FUNCTION_BLOCK "fbUO_MX_SETUP"
TITLE = UO : MX_SETUP
{ S7_Optimized_Access := 'TRUE' }
AUTHOR : REO
NAME : MX_SETUP
VERSION : 2.0
//****************************************************************************************************
// Code generated by SFC Generator V1.13 on 23/11/18 15:00:24 by  David Paspa from File G:\Business\Synertec\MPI.SMS\automation\code\awlMaster\stencil\seq_hdr.awl
//****************************************************************************************************
//****************************************************************************************************
//================================ SEQ HEADER ================================//
//            Copyright 2018 Rieckermann Engineering Operations               //
//----------------------------------------------------------------------------//
// Title: UO_MX_SETUP                                                       //
//                                                                            //
// Description:                                                               //
// Unit Operation for setup of equipment for manufacturing operations.                                                        //
//                                                                            //
// // SFC Revision History:
// Rev By               Date        CC         Note
// 2.0 David Paspa      09-Aug-2018            Reboot for S7-1500.
// 0.1 Gerald Kontriner 14-Sep-2009            SFC structural design                                                       //
//----------------------------------------------------------------------------//
// Sequencer Revision History:                                                //
// Rev By               Date        CC        Note                            //
// 2.0 David Paspa      05-Jan-2018 NA        Reboot for S7-1500.             //
// 1.6 Khairul Basar    19-Nov-2009 NA        Reset #sqSequencer.STEP.Active  //
//                                            when STEP Finished.             //
// 1.5 Khairul Basar    15-Oct-2009 NA        Placeholder inserted:           //
//                                            "udtSQ_UO";          //
// 1.4 Khairul Basar    06-Oct-2009 NA        R #PAUSE;                       //
// 1.3 Khairul Basar    30-Sep-2009 NA        SEQ_HDR change STEP-0 code      //
//                                            deleted.                        //
// 1.2 Khairul Basar    26-Sep-2009 NA        Refer R4.                       //
// 1.1 Khairul Basar    23-Sep-2009 NA        Refer R3.                       //
// 1.0 Khairul Basar    20-Sep-2009 NA        STEP.Finished flag reset by     //
//                                            JUMP_MAN.                       //
// 0.9 Khairul Basar    11-Sep-2009 NA        SQ_TIMER added as VAR, declared //
//                                            in SEQ_FTR.                     //
// 0.8 Khairul Basar    09-Sep-2009 NA        SqSequencer.Err_Fault is reset  //
//                                            on Stop cmd, Step-0 dead code   //
//                                            deleted from ACT & Verify.      //
//                                            STP_FTR Step_withErr flag       //
//                                            STEP_NUM place holder           //
//                                            configured.                     //
// 0.7 Khairul Basar    28-Aug-2009 NA        SQ_FINISHED OUT added again.    //
//                                            Deleted during major mod R3.    //
// 0.6 Khairul Basar    23-Aug-2009 NA        Refer R2.                       //
// 0.5 Khairul Basar    23-Aug-2009 NA        Refer R1.                       //
// 0.4 Khairul Basar    18-Aug-2009 NA        Reset Step done with/out error  //
//                                            bits using FC:RSET.             //
// 0.3 David Paspa      16-Aug-2009 NA        Added placeholders for header   //
//                                            name and version and revision   //
//                                            history.                        //
// 0.2 Khairul Basar    11-Aug-2009 NA        Retired external udt file for   //
//                                            Static type parameters. All     //
//                                            parameters now IN, OUT or       //
//                                            IN_OUT.                         //
// 0.1 Khairul Basar    12-Jun-2009 NA        Initial design.                 //
//----------------------------------------------------------------------------//
// R4:                                                                        //
// 1.If SQ not finished Resume command will start Step timer, and redo the    //
// last action, verify the feedback.                                          //
// 2."STEP.finished" flag is ANDed with "TRN_AND_JUMP" in the snippet file    //
// TRN_HDR.This is to avoid checking of transition logic if STEP is not       //
// finished yet.                                                              //
// 3.MDCH, Load & transfer typo corrected.                                    //
//                                                                            //
// R3:                                                                        //
// 1.SqStepTimer.IN is reset in STEP_FTR instead of resetting it in TRN_HDR.  //
// This is because TRN_HDTR is not included in the Last step and StepTimer    //
// must reset in the last step.                                               //
// 2.Reset all the timers when SQ stops.Reset done in SEQ_HDR.                //
// Also STEP-finished flag reset when SQ is OFF to                            //
// scan last step.                                                            //
//                                                                            //
// R2:                                                                        //
// 1.Any step error will send the Sequencer into Pause state.Code added in    //
// SEQ_HDR.Snippet Place holder for Bool-array 24 is   //
// deleted.                                                                   //
//                                                                            //
// R1:                                                                        //
// 1.sqStepTimer:All Verification Code must satisfy the condition finish step //
// action within STEP_DELAY time(40s).If step actions not finished within the //
// time period the error flag will raise High signal.Else timer will reset.   //
// 2.sqRunTimer Added therefore can be used as retentive & non retentive.     //
// 3.sqSequencer: This is re-structured UDT which is redefined the symbol     //
// names as well as it gives more clearity.                                   //
// 4.fcMODE and fcCMD functions are added to handle the mode & command        //
// independently regardless of other logic.Two separate UDT udtMODE & udt     //
// CMD assigned to Mode & command function respectively.                      //
// 5.MAN_JUMP programed for manual mode jump operation with or without        //
// Transition code satisfied.TRN_AND_JUMP & NO_VERIFC are the parameters      //
// which will define whether verification code & transition code need to be   //
// checked to perform jump operation.                                         //
// 6.Auto to Manual switchover will be bumpless & will not affect step        //
// operation.Manual to auto switchover can be used to resume Step action at   //
// defined.                                                                   //
// Step number entered in STEPNO_JUMP.                                        //
//                                                                            //
// Parameters:                                                                //
// INPUTS                                                                     //
// ======                                                                     //
// SQ_CMD          Sequence command input inherited from object block         //
//                 0: off/idle                                                //
//                 1: start/initiate                                          //
//                 2: pause                                                   //
//                 3: resume                                                  //
//                 4: reserved (not programmed)                               //
//                 5: reserved (not programmed)                               //
//                 6: abort/go to last step                                   //
//                 7: acknowledge error/fault                                 //
// SQ_MODE         Sequencer Auto/Manual input inherited from object block    //
//                 1: manual                                                  //
//                 2: auto                                                    //
//                                                                            //
// INPUT/OUTPUTS                                                              //
// =============                                                              //
// SQ_JUMP_MAN     Allows manual jumping from one step to the next step. The  //
//                 manual jump flag is ORed with the transition process       //
//                 condition and so can be used to bypass the condition if the//
//                 sequence will not progress.                                //
//                 This input can also be used to jump to any step even       //
//                 when no transition -> step linkage exists. This is only    //
//                 possible when the SQ_MODE is in manual and SQ is in the    //
//                 idle step. The step to jump to is specified in             //
//                 SQ_man_jump_to_step (not accesseble by this FB in/out      //
//                 interface but a separate DB memory location).              //
//                                                                            //
// OUTPUTS                                                                    //
// =======                                                                    //
// SQ_STATE        The calculated state of the sequence                       //
//                 0: off/idle                                                //
//                 1: start/initiated                                         //
//                 2: paused                                                  //
//                 3: resumed                                                 //
//                 4: reserved (wrong Mode)                                   //
//                 5: reserved (Wrong commad)                                 //
//                 6: aborted/go to last step                                 //
//                 7: acknowledged error/fault                                //
// CURSTEP         Current step being proccessed.                             //
// S_ACTIVE        If current step is active                                  //
// NXT_STEP        Next step to jump to if transition condition is true       //
// ERR_FAULT       True if any error/ or fault present                        //
// PAUSED          True if step is paused                                     //
// OFF_IDLE        Sequence is not running but ready for next SQ (in step=0)  //
//----------------------------------------------------------------------------//
// Define variables:                                                          //
//----------------------------------------------------------------------------//
   VAR_IN_OUT
      _emm_vessel_mi_vessel_pv : Real;   // Vessel measured mass
      _emx_drain_state : Int;   // State for MX drain valves
      _emv_inlet_state : Int;   // Sprayball inlet state
      _emt_hex_state : Int;   // Heat exchanger temperature control state
      _vessel_mx : Int;   // Manufacturing vessel selection M1 or M2
      _emc_gas_pi_vessel_pv : Real;   // Vessel pressure
      _vacuum_hold_test : Bool;   // Vacuum hold test enquiry
      _emm_vessel_state : Int;   // Device State of emm_vessel
      _emc_water_state : Int;   // Device State of emc_water
      _emx_mmfl_state : Int;   // Device State of emx_mmfl
      _emv_vessel_state : Int;   // Device State of EVxy04
      _emg_filter_state : Int;   // Device State of emg_filter
      _emx_transfer_state : Int;   // Device State of emx_transfer
      _emc_gas_state : Int;   // Device State of emc_gas
      _emx_drain_subs : Int;   // Substate for MX drain valves
      _emx_drain_cmd : Int;   // Command for MX drain valves
      _emv_inlet_subs : Int;   // Sprayball inlet substate
      _emv_inlet_cmd : Int;   // Sprayball inlet command
      _emt_hex_cmd : Int;   // Heat exchanger temperature control command
      _emt_hex_subs : Int;   // Heat exchanger temperature control substate
      _emt_hex_drain_time : Time;   // Heat exchanger drain time
      _emc_gas_medium_gas : Int;   // Medium selection for emc_gas
      _emm_vessel_cmd : Int;   // Command to emm_vessel
      _emm_vessel_subs : Int;   // Substate selection to emm_vessel
      _emc_water_cmd : Int;   // Command to emc_water
      _emc_water_subs : Int;   // Substate selection to emc_water
      _emc_water_medium_liquid : Int;   // Medium selection for emc_water
      _emx_mmfl_cmd : Int;   // Command to emx_mmfl
      _emv_vessel_subs : Int;   // Substate selection to emv_vessel
      _emx_mmfl_subs : Int;   // Substate selection to emx_mmfl
      _emv_vessel_cmd : Int;   // Command to emv_vessel
      _emx_transfer_cmd : Int;   // Command to emx_transfer
      _emg_filter_cmd : Int;   // Command to emg_filter
      _emx_transfer_subs : Int;   // Substate selection to EXxy07
      _emg_filter_subs : Int;   // Substate selection to emg_filter
      _emc_gas_cmd : Int;   // Command to emc_gas
      _emc_gas_subs : Int;   // Substate selection to emc_gas
      dummy : Bool;   // Dummy placeholder for call without comma
   END_VAR

   VAR
      smc : "udtModeCommandSFC";   // SFC mode and command
      sqStepTimer {OriginalPartName := 'IEC_TIMER'; LibVersion := '1.0'} : TON_TIME;
      sqRunTimer : "fbRunTimer";
      sqSequencer : "udtSFCSequence32";
      SQ_TIMER {OriginalPartName := 'IEC_TIMER'; LibVersion := '1.0'} : TON_TIME;
      SQ_TIMER2 {OriginalPartName := 'IEC_TIMER'; LibVersion := '1.0'} : TON_TIME;
      SQ_TIMER3 {OriginalPartName := 'IEC_TIMER'; LibVersion := '1.0'} : TON_TIME;
      sqSeqTimerStart : Bool;
      sqSeqTimerStart2 : Bool;
      sqSeqTimerStart3 : Bool;
      sqSeqTimerElapsed : Time;
      sqSeqTimerElapsed2 : Time;
      sqSeqTimerElapsed3 : Time;
      sqSeqTimerExpired : Bool;
      sqSeqTimerExpired2 : Bool;
      sqSeqTimerExpired3 : Bool;
      sqStepTimerElapsed : Time;
      sqStepTimerExpired : Bool;
      _r_time_hex_drain : Time;   // MX SETUP Heat exchanger drain time
      _real_not_held : Real;   // UO_MX_SETUP Vacuum pressure hold test failed
      _real_vacuum_fail : Real;   // UO_MX_SETUP Vacuum failed pressure after vacuum timer expired
      _log_real_pressure_mx : Bool;   // UO_MX_SETUP Vessel pressure
      _real_pressure_mx : Real;   // UO_MX_SETUP Vessel pressure
      _log_real_not_held : Bool;   // UO_MX_SETUP Vacuum pressure hold test failed
      _vacuum_held_begin_time : Time_Of_Day;   // vacuum hold begin time
      _vacuum_held_end_time : Time_Of_Day;   // vacuum hold end time
      _time_act_vacuum_held : Time;   // UO_MX_SETUP Vacuum held time
      _log_time_act_vacuum_held : Bool;   // UO_MX_SETUP Vacuum held time
      _prompt_not_held : Bool;   // UO_MX_SETUP Operator to confirm to retry as vacuum pressure not held
      _prompt_not_held_confirm_yes : Bool;   // UO_MX_SETUP Operator to confirm to retry vacuum pressure not held confirmed yes
      _prompt_not_held_confirm_no : Bool;   // UO_MX_SETUP Operator to confirm to retry vacuum pressure not held confirmed no
      _log_msg_not_held_repeat : Bool;   // UO_MX_SETUP Operator confirmed to retry when vacuum pressure not held
      _log_msg_not_held_abort : Bool;   // UO_MX_SETUP Operator confirmed to abort when vacuum pressure not held
      _prompt_not_reach : Bool;   // UO_MX_SETUP Operator to confirm retry when vacuum pressure not reached setpoint
      _prompt_not_reach_confirm_yes : Bool;   // UO_MX_SETUP Operator confirmed retry when vacuum pressure not reached setpoint
      _prompt_not_reach_confirm_no : Bool;   // UO_MX_SETUP Operator confirmed abort when vacuum pressure not reached setpoint
      _log_msg_not_reach_repeat : Bool;   // UO_MX_SETUP Operator confirmed retry when vacuum pressure not reached setpoint
      _log_msg_not_reach_abort : Bool;   // UO_MX_SETUP Operator confirmed abort when vacuum pressure not reached setpoint
      _log_real_vacuum_fail : Bool;   // UO_MX_SETUP Vacuum failed after vacuum timer expired
      _log_msg_vacuum_begin : Bool;   // UO_MX_SETUP Vacuum begin time
      _log_msg_setup_end : Bool;   // UO_MX_SETUP end time
      _log_msg_setup_begin : Bool;   // UO_MX_SETUP begin time
      _r_pres_vac_fail : Real;   // MX SETUP Vacuum hold test fail pressure
      _r_pres_vac : Real;   // MX SETUP Vacuum setpoint
      _r_time_vac_hold : Time;   // MX SETUP Time for vacuum hold test
      _r_time_eject : Time;   // MX SETUP Time to run vacuum system before timeout
      _prompt_connect_ok_confirm_yes : Bool;   // UO_MX_SETUP Operator confirm vessel connections made confirmed yes
      _prompt_connect_ok : Bool;   // UO_MX_SETUP Operator to confirm all vessel connections are properly made
   END_VAR


BEGIN
NETWORK
TITLE = Call Mode checking function
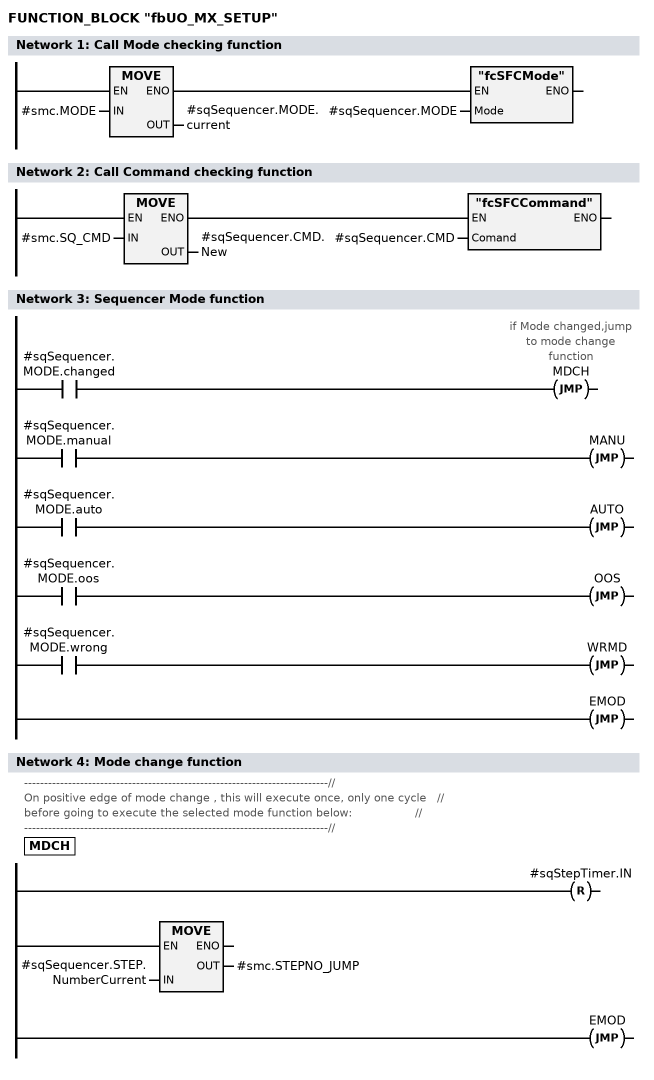
      L #smc.MODE;
      T #sqSequencer.MODE.current;
      CALL "fcSFCMode"
      (  Mode                        := #sqSequencer.MODE
      );

NETWORK
TITLE = Call Command checking function
      L #smc.SQ_CMD;
      T #sqSequencer.CMD.New;
      CALL "fcSFCCommand"
      (  Comand                      := #sqSequencer.CMD
      );

NETWORK
TITLE = Sequencer Mode function

      A #sqSequencer.MODE.changed;
      JC MDCH;// if Mode changed,jump to mode change function
      A #sqSequencer.MODE.manual;
      JC MANU;
      A #sqSequencer.MODE.auto;
      JC AUTO;
      A #sqSequencer.MODE.oos;
      JC OOS;
      A #sqSequencer.MODE.wrong;
      JC WRMD;
      JU EMOD;

NETWORK
TITLE = Mode change function
//----------------------------------------------------------------------------//
// On positive edge of mode change , this will execute once, only one cycle   //
// before going to execute the selected mode function below:                  //
//----------------------------------------------------------------------------//
MDCH:      NOP 0;
      SET;
      R #sqStepTimer.IN;
      L #sqSequencer.STEP.NumberCurrent;
      T #smc.STEPNO_JUMP;
      JU EMOD;

NETWORK
TITLE = Manual Mode function
//----------------------------------------------------------------------------//
// #TRN_AND_JUMP=can set/reset                                                //
// #sqSequencer.STEP.JumpCtrl=Can set/reset by #MAN_JUMP                      //
// #NO_VERIFIC=Can set/ Reset                                                 //
//----------------------------------------------------------------------------//
MANU:      NOP 0;//Manual mode selected



      A #smc.MAN_JUMP;
      = #sqSequencer.STEP.JumpCtrl;
      A #smc.MAN_JUMP;
      JCN EMOD;

      L #smc.STEPNO_JUMP;
      T #sqSequencer.STEP.NumberNext;
      T #sqSequencer.STEP.NumberCurrent;
      R #smc.MAN_JUMP;//Reset MAN_JUMP after loading user destination Step number
      R #sqSequencer.STEP.Finished;//Reset finish flag, to execute next step action
      JU EMOD;

NETWORK
TITLE = Auto Mode function
//----------------------------------------------------------------------------//
// #TRN_AND_JUMP=always set                                                   //
// #sqSequencer.STEP.JumpCtrl=Always set                                      //
// #NO_VERIFIC=Alwasy Reset                                                   //
//----------------------------------------------------------------------------//
AUTO:      NOP 0;//Auto mode selected



      R #smc.MAN_JUMP;
      S #smc.TRN_AND_JUMP;
      R #smc.NO_VERIFIC;
      S #sqSequencer.STEP.JumpCtrl;//Always Set in auto mode

      L #sqSequencer.STEP.NumberCurrent;
      T #smc.STEPNO_JUMP;
      JU EMOD;
NETWORK
TITLE = OOS mode function

OOS:      NOP 0;// Out of service
      JU EMOD;
WRMD:      NOP 0;//Wrong mode selected
      S #sqSequencer.Error_Fault;
      L "dbCONST".SEQ.STATE.WRMODE;
      T #smc.SQ_STATE;

      JU EMOD;

NETWORK
TITLE = Mode not changedd

      NOP 0;

NETWORK
TITLE = End Mode function

EMOD:      NOP 0;

NETWORK
TITLE = An error will Pause the Sequencer,Operator must Resume SQ to run

      A #sqSequencer.Error_Fault;
      AN #sqSequencer.CMD.Changed;
      JC PAUS;

NETWORK
TITLE = Command Action function

      A #sqSequencer.CMD.Changed;
      JCN CNCH;// if Command not changed,jump to end function
      R #sqStepTimer.IN;

      A #sqSequencer.CMD.Start;
      JC STRT;

      A #sqSequencer.CMD.Stop;
      JC STOP;

      A #sqSequencer.CMD.Pause;
      JC PAUS;

      A #sqSequencer.CMD.Resume;
      JC RESM;

      A #sqSequencer.CMD.Abort;
      JC _abrt_begin;

      A #sqSequencer.CMD.Ack;
      JC ACKN;

      A #sqSequencer.CMD.wrong;
      JC WCMD;

      JU ECMD;//Wrong command/not specified command
//End Comand function

NETWORK
TITLE = Comand -Start/Initiate action function

STRT:      NOP 0;
      R #smc.OFF_IDLE;
      R #smc.ABORTED;
      R #smc.PAUSED;
      R #sqSequencer.STEP.Active;
      R #sqSequencer.STEP.Finished;
      R #sqSequencer.STEP.ActionFinished;
      R #sqSequencer.STEP.Jump;
      R #sqSequencer.STEP.TimerExpired;
      R #sqSequencer.STEP.Error_Fault;
      R #sqSequencer.STEP.ActionVerified;
      R #sqStepTimer.IN;

//      S     #sqRunTimer.RESET;

//----------------------------------------------------------------------------//
// Load Initial step Number:                                                  //
//----------------------------------------------------------------------------//
      L 1;
      T #sqSequencer.STEP.Initial;
      L #sqSequencer.STEP.Initial;
      T #sqSequencer.STEP.NumberCurrent;
      T #sqSequencer.STEP.NumberNext;

      L "dbCONST".SEQ.STATE.STARTED;
      T #smc.SQ_STATE;

NETWORK
TITLE = Reset sequence Done bits
//------------------------------------------------------------------------//
// Reset Step done bits:                                                  //
//------------------------------------------------------------------------//
      CALL FILL_BLK
      {value_type := 'Bool', count_type := 'UInt'}
      (  IN                          := 0 ,
         COUNT                       := 32 ,
         OUT                         := #sqSequencer.STEP.Done[1]
      );

NETWORK
TITLE = Reset sequence Error bits
//------------------------------------------------------------------------//
// Reset Step error bits:                                                 //
//------------------------------------------------------------------------//
      CALL FILL_BLK
      {value_type := 'Bool', count_type := 'UInt'}
      (  IN                          := 0 ,
         COUNT                       := 32 ,
         OUT                         := #sqSequencer.STEP.WithError[1]
      );

      JU ECMD;//End Function

NETWORK
TITLE = Comand -Stop action function

STOP:      NOP 0;
      S #smc.OFF_IDLE;
      R #sqSequencer.STEP.Active;
      R #sqSequencer.STEP.Finished;
      R #sqSequencer.STEP.ActionFinished;
      R #sqSequencer.STEP.Jump;
      R #sqSequencer.STEP.TimerExpired;
      R #sqSequencer.STEP.Error_Fault;
      R #sqSequencer.Error_Fault;
      R #sqSequencer.STEP.ActionVerified;
      R #sqRunTimer.ENABLE;
      R #sqStepTimer.IN;
      R #sqSeqTimerStart;
      R #sqSeqTimerStart2;
      R #sqSeqTimerStart3;
      R #smc.PAUSED;
      R #smc.ABORTED;


//Go to last step
      L 18;
      T #sqSequencer.FinalStep;
      T #sqSequencer.STEP.NumberNext;

      JU ECMD;//End Function

NETWORK
TITLE = Comand -Pause action function

PAUS:      NOP 0;
      S #smc.PAUSED;
      R #smc.S_ACTIVE;
      S #sqRunTimer.PAUSE;
      L #sqSequencer.STEP.NumberCurrent;
      T #smc.STEPNO_JUMP;
      L "dbCONST".SEQ.STATE.PAUSED;
      T #smc.SQ_STATE;

      JU ECMD;//End Function

NETWORK
TITLE = Comand -Resume action function

RESM:      NOP 0;
      R #smc.PAUSED;
      R #sqRunTimer.PAUSE;
      R #sqStepTimer.IN;//Reset Step timer
      L "dbCONST".SEQ.STATE.RESUMED;
      T #smc.SQ_STATE;

      A #smc.SQ_FINISHED;
      JC ECMD;
      R #sqSequencer.STEP.Active;
      R #sqSequencer.STEP.Finished;
      R #sqSequencer.STEP.ActionFinished;

      JU ECMD;//End Function

NETWORK
TITLE = Comand -Abort action function

_abrt_begin:      NOP 0;

      S #smc.ABORTED;
      R #sqSequencer.STEP.Active;
      R #sqSequencer.STEP.Finished;
      R #sqSequencer.STEP.ActionFinished;
      R #sqSequencer.STEP.Jump;
      R #sqSequencer.STEP.TimerExpired;
      R #sqSequencer.STEP.Error_Fault;
      R #sqSequencer.Error_Fault;
      R #sqSequencer.STEP.ActionVerified;
      R #sqRunTimer.ENABLE;
      R #sqStepTimer.IN;
      R #sqSeqTimerStart;
      R #sqSeqTimerStart2;
      R #sqSeqTimerStart3;
      R #smc.PAUSED;
      R #smc.OFF_IDLE;


//Go to last step
      L 18;
      T #sqSequencer.FinalStep;
      T #sqSequencer.STEP.NumberNext;

      JU ECMD;

NETWORK
TITLE = Comand -Acknowledge action function

ACKN:      NOP 0;
      R #smc.ERR_FAULT;
      R #sqSequencer.Error_Fault;
      L "dbCONST".SEQ.STATE.ACKNOWLEDGED;
      T #smc.SQ_STATE;

      JU ECMD;//End Function

NETWORK
TITLE = Comand -wrong/unavailable

WCMD:      NOP 0;

      S #sqSequencer.Error_Fault;
      L "dbCONST".SEQ.STATE.WRCMD;
      T #smc.SQ_STATE;

      JU ECMD;
NETWORK
TITLE = Comand -not changedd

CNCH:      NOP 0;// Command not changed

NETWORK
TITLE = End command Function

ECMD:      NOP 0;

NETWORK
TITLE = Sequencer Step Jump distrubution list
//------------------------------------------------------------------------//
// Sequencer step jump list. Load the step number to execute the step:    //
//------------------------------------------------------------------------//
      L #sqSequencer.STEP.NumberCurrent;
      JL SQER;// If Sequencer Step number invalid or greater than available number of step
      JU S000;// Exceptional Error Handling
      JU S001;// STEP-001:
      JU S002;// STEP-002:
      JU S003;// STEP-003:
      JU S004;// STEP-004:
      JU S005;// STEP-005:
      JU S006;// STEP-006:
      JU S007;// STEP-007:
      JU S008;// STEP-008:
      JU S009;// STEP-009:
      JU S010;// STEP-010:
      JU S011;// STEP-011:
      JU S012;// STEP-012:
      JU S013;// STEP-013:
      JU S014;// STEP-014:
      JU S015;// STEP-015:
      JU S016;// STEP-016:
      JU S017;// STEP-017:
      JU S018;// STEP-018:


  //------------------------------------------------------------------------//
  // If Step number is Invalid or Out of Range:                             //
  //------------------------------------------------------------------------//
SQER:      NOP 0;
      A "alwaysLow";
      S #sqSequencer.Error_Fault;
      JU COMM;// Jump to Common Sequencer code handling function

NETWORK
TITLE = STEP0 STEP0 STEP0 STEP0 STEP0 STEP0 STEP0 STEP0 STEP0 STEP0 STEP
//------------------------------------------------------------------------//
// STEP0 STEP0 STEP0 STEP0 STEP0 STEP0 STEP0 STEP0 STEP0 STEP0 STEP0 STEP //
// AUTOCODE   AUTOCODE   AUTOCODE   AUTOCODE   AUTOCODE   AUTOCODE   AUTO //
// STEP0 STEP0 STEP0 STEP0 STEP0 STEP0 STEP0 STEP0 STEP0 STEP0 STEP0 STEP //
//------------------------------------------------------------------------//

NETWORK
TITLE = S000: STEP0::If Paused exit

S000:      NOP 0;
      JU COMM;






NETWORK
TITLE = S001: STEP-01::UO_MX_SETUP : Setup Unit Operation Commenced
//================================ STEP HEADER ===========================//
// STEP001 STEP001 STEP001 STEP001
// AUTOCODE   AUTOCODE   AUTOCODE   AUTOCODE   AUTOCODE   AUTOCODE   AUTO //
// STEP001 STEP001 STEP001 STEP001
//------------------------------------------------------------------------//
// Log Mx SETUP operation begin time.
// Prompt operator to confirm that all vessel connections, including the permanent flexible connections are properly made.
//
// Start EMX1_SETUP_CIPSIP to connect MMFLx to Drain.
//------------------------------------------------------------------------//
S001:      NOP 0;

      SET;
      R #sqSequencer.STEP.jumpDone[01];
      A #sqSequencer.CMD.Pause;//If paused jump
      JC COMM;

NETWORK
TITLE = S001:STEP-01:Begin Action

      A #sqSequencer.STEP.Finished;
      JC A001;// Exit Action code, Jump to A001 Transition code

    //----------------------------------------------------------------------//
    // Begin step Action:                                                   //
    //----------------------------------------------------------------------//
      A #sqSequencer.STEP.Active;
      JC L001;// Action number loaded, Jump to L001--Step Action List

    //----------------------------------------------------------------------//
    // Load Default/Initial Step action number:                             //
    //----------------------------------------------------------------------//
      S #sqSequencer.STEP.Active;
      S #sqStepTimer.IN;
      L 1;//First Action, Step must contain Minimum one action
      T #sqSequencer.STEP.ActionNumber;

//----------------------------------------------------------------------------//
// Step action list.                                                          //
// aann=mini Action step number(aa) inside main step number(nn)               //
// First Action aa00, Second action ab00, Third ac00, etc.                    //
//----------------------------------------------------------------------------//
L001:      NOP 0;

      L #sqSequencer.STEP.ActionNumber;
      JL r001;//Wrong Action number
      JU _001;//Action error handling
      JU aa01;//ACTION-01
      JU ab01;//ACTION-02


//----------------------------------------------------------------------------//
// More step action in the list can be inserted here, upto ab is tested:      //
//----------------------------------------------------------------------------//
r001:      NOP 0;//Wrong action number
      S #sqSequencer.Error_Fault;
      JU k001;//Exit
_001:      NOP 0;// Action error handling
      JU k001;// Exit






NETWORK
TITLE = S001:: STEP-001:: : ACTION CODE
//================================ ACT HEADER ============================//
// ACTION ACTION ACTION ACTION ACTION ACTION ACTION ACTION ACTION ACTION  //
// AUTOCODE   AUTOCODE   AUTOCODE   AUTOCODE   AUTOCODE   AUTOCODE   AUTO //
// ACTION ACTION ACTION ACTION ACTION ACTION ACTION ACTION ACTION ACTION  //
//------------------------------------------------------------------------//
// //Reset the MMFL transfer line EM
aa01:      NOP 0;

  //------------------------------------------------------------------------//
  // ACT ACT ACT ACT ACT ACT ACT ACT ACT ACT ACT ACT ACT ACT ACT ACT ACT    //
  //------------------------------------------------------------------------//
      L "dbCONST".BLK.CMD.STOP;
      T #_emx_mmfl_cmd;

  //------------------------------------------------------------------------//
  // VERIFY  VERIFY VERIFY VERIFY VERIFY VERIFY VERIFY VERIFY VERIFY VERIFY //
  //------------------------------------------------------------------------//
      A(;
      L #_emx_mmfl_state;
      L "dbCONST".BLK.STATE.STOPPED;
      ==I;
      );
      S #sqSequencer.STEP.ActionVerified;//Action verified

  //------------------------------------------------------------------------//
  // Action done:                                                           //
  //------------------------------------------------------------------------//
      O #sqSequencer.STEP.ActionVerified;
      O #smc.NO_VERIFIC     ;//No verification , bypass verification code
      S #sqSequencer.STEP.ActionFinished;






  //============================= ACT FOOTER ===============================//
  // AUTOCODE   AUTOCODE   AUTOCODE   AUTOCODE   AUTOCODE   AUTOCODE   AUTO //
  // Get Ready after action finished:                                       //
  //------------------------------------------------------------------------//
      A #sqSequencer.STEP.ActionFinished;
      JCN k001;

  //------------------------------------------------------------------------//
  // Reset Action finished flag, ready for next step action:                //
  //------------------------------------------------------------------------//
      R #sqSequencer.STEP.ActionVerified;
      R #sqSequencer.STEP.ActionFinished;

  //------------------------------------------------------------------------//
  // Load Next Step Action number:                                          //
  //------------------------------------------------------------------------//
      L 02;//Load next Action
      T #sqSequencer.STEP.ActionNumber;






NETWORK
TITLE = S001:: STEP-001:: : ACTION CODE
//================================ ACT HEADER ============================//
// ACTION ACTION ACTION ACTION ACTION ACTION ACTION ACTION ACTION ACTION  //
// AUTOCODE   AUTOCODE   AUTOCODE   AUTOCODE   AUTOCODE   AUTOCODE   AUTO //
// ACTION ACTION ACTION ACTION ACTION ACTION ACTION ACTION ACTION ACTION  //
//------------------------------------------------------------------------//
// //Log Mx SETUP operation begin time.
// //Prompt operator to confirm correct vessel connections.
// //Start EMX1_SETUP_CIPSIP
ab01:      NOP 0;

  //------------------------------------------------------------------------//
  // ACT ACT ACT ACT ACT ACT ACT ACT ACT ACT ACT ACT ACT ACT ACT ACT ACT    //
  //------------------------------------------------------------------------//
  //Log CIPSIP operation begin
      SET;
      S #_log_msg_setup_begin;

      SET;
      S #_prompt_connect_ok;

//Start EMX1_CIPSIP_SETUP.
      L "dbCONST".BLK.EMX1.SUBS.SETUP_CIPSIP;
      T #_emx_mmfl_subs;
      L "dbCONST".BLK.CMD.START;
      T #_emx_mmfl_cmd;

  //------------------------------------------------------------------------//
  // VERIFY  VERIFY VERIFY VERIFY VERIFY VERIFY VERIFY VERIFY VERIFY VERIFY //
  //------------------------------------------------------------------------//
      A(;
      L #_emx_mmfl_subs;
      L "dbCONST".BLK.EMX1.SUBS.SETUP_CIPSIP;
      ==I;
      );
      S #sqSequencer.STEP.ActionVerified;//Action verified

  //------------------------------------------------------------------------//
  // Action done:                                                           //
  //------------------------------------------------------------------------//
      O #sqSequencer.STEP.ActionVerified;
      O #smc.NO_VERIFIC     ;//No verification , bypass verification code
      S #sqSequencer.STEP.ActionFinished;






  //============================= STEP FOOTER ==============================//
  // AUTOCODE   AUTOCODE   AUTOCODE   AUTOCODE   AUTOCODE   AUTOCODE   AUTO //
  // Get Ready after action finished:                                       //
  //------------------------------------------------------------------------//
      A #sqSequencer.STEP.ActionFinished;
      JCN k001;

  //------------------------------------------------------------------------//
  // Reset Action finished flag, ready for next step action:                //
  //------------------------------------------------------------------------//
      R #sqSequencer.STEP.ActionVerified;
      R #sqSequencer.STEP.ActionFinished;

  //------------------------------------------------------------------------//
  // If ALL actions are finished:                                           //
  //------------------------------------------------------------------------//
      SET;
      S #sqSequencer.STEP.Finished;
      R #sqSequencer.STEP.Active;
      S #sqSequencer.STEP.Done[01];

  //------------------------------------------------------------------------//
  // End Step action(s):                                                    //
  //------------------------------------------------------------------------//
      JU k001;

//----------------------------------------------------------------------------//
// Finished Step Action(s):                                                   //
//----------------------------------------------------------------------------//
k001:      NOP 0;

      A #sqStepTimerExpired;
      S #sqSequencer.STEP.WithError[01];// Step error flag
      S #sqSequencer.Error_Fault;
      R #sqStepTimer.IN;

NETWORK
TITLE = S001:STEP-001::Begin Transition
//------------------------------------------------------------------------//
// Begin the transition code:                                             //
//------------------------------------------------------------------------//
A001:      NOP 0;
      R #sqStepTimer.IN;






  //============================= TRAN HEADER ==============================//
  // AUTOCODE   AUTOCODE   AUTOCODE   AUTOCODE   AUTOCODE   AUTOCODE   AUTO //
  // Bypass transition if manual jump:                                      //
  //------------------------------------------------------------------------//
      A #sqSequencer.STEP.Finished;
      A #smc.TRN_AND_JUMP   ;//Manual jump is set Transition as bypassed
      JCN COMM            ;//exit

NETWORK
TITLE = S001::STEP 001:TRAN 001: Confirmation received.
//----------------------------------------------------------------------------//
// TRAN   TRAN   TRAN   TRAN   TRAN   TRAN   TRAN   TRAN   TRAN   TRAN   TRAN //
// TRAN   TRAN   TRAN   TRAN   TRAN   TRAN   TRAN   TRAN   TRAN   TRAN   TRAN //
//----------------------------------------------------------------------------//
// Confirmation from operator received and CIPSIP_SETUP finished.
//----------------------------------------------------------------------------//
// CONDITION   CONDITION   CONDITION   CONDITION   CONDITION   CONDITION   CO //
// CONDITION   CONDITION   CONDITION   CONDITION   CONDITION   CONDITION   CO //
//----------------------------------------------------------------------------//
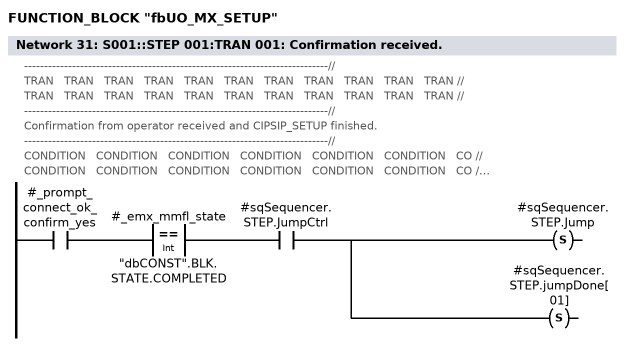
      A #_prompt_connect_ok_confirm_yes;
      A(;
      L #_emx_mmfl_state;
      L "dbCONST".BLK.STATE.COMPLETED;
      ==I;
      );






  //============================= TRAN FOOTER ==============================//
  // Transition jump control:                                               //
  //------------------------------------------------------------------------//
      A #sqSequencer.STEP.JumpCtrl;
      S #sqSequencer.STEP.Jump;
      S #sqSequencer.STEP.jumpDone[01];

NETWORK
TITLE = S001:t001::TRANS-v: EXIT TRANSITION AND READY THE NEXT STEP
//------------------------------------------------------------------------//
// Check the jump flag and jump to the next step if the transition        //
// condition is true and has set the jump flag:                           //
//------------------------------------------------------------------------//
      A #sqSequencer.STEP.Jump;
      JCN x001;

      R #sqSequencer.STEP.Jump;
      R #sqSequencer.STEP.Finished;

      L 02   ;// Load next STEPNO to jump to if transition satisfied
      T #sqSequencer.STEP.NumberNext;//Next Step02.

      JU COMM            ;// Transition satisfied, Exit, go to next step
x001:      NOP 0;






NETWORK
TITLE = S001::STEP-001:EXIT TRANSITION:
//========================== STEP TRANSFER ===============================//
// Jump to the common step progression code:                              //
//------------------------------------------------------------------------//
      JU COMM;






NETWORK
TITLE = S002: STEP-02::UO_MX_SETUP : Setup for PW and drain heat exchanger
//================================ STEP HEADER ===========================//
// STEP002 STEP002 STEP002 STEP002
// AUTOCODE   AUTOCODE   AUTOCODE   AUTOCODE   AUTOCODE   AUTOCODE   AUTO //
// STEP002 STEP002 STEP002 STEP002
//------------------------------------------------------------------------//
// Set emc_water to substate SETUP with MEDIUM PW.
//
// Drain the heat exchanger.
//------------------------------------------------------------------------//
S002:      NOP 0;

      SET;
      R #sqSequencer.STEP.jumpDone[02];
      A #sqSequencer.CMD.Pause;//If paused jump
      JC COMM;

NETWORK
TITLE = S002:STEP-02:Begin Action

      A #sqSequencer.STEP.Finished;
      JC A002;// Exit Action code, Jump to A002 Transition code

    //----------------------------------------------------------------------//
    // Begin step Action:                                                   //
    //----------------------------------------------------------------------//
      A #sqSequencer.STEP.Active;
      JC L002;// Action number loaded, Jump to L002--Step Action List

    //----------------------------------------------------------------------//
    // Load Default/Initial Step action number:                             //
    //----------------------------------------------------------------------//
      S #sqSequencer.STEP.Active;
      S #sqStepTimer.IN;
      L 1;//First Action, Step must contain Minimum one action
      T #sqSequencer.STEP.ActionNumber;

//----------------------------------------------------------------------------//
// Step action list.                                                          //
// aann=mini Action step number(aa) inside main step number(nn)               //
// First Action aa00, Second action ab00, Third ac00, etc.                    //
//----------------------------------------------------------------------------//
L002:      NOP 0;

      L #sqSequencer.STEP.ActionNumber;
      JL r002;//Wrong Action number
      JU _002;//Action error handling
      JU aa02;//ACTION-01
      JU ab02;//ACTION-02
      JU ac02;//ACTION-03


//----------------------------------------------------------------------------//
// More step action in the list can be inserted here, upto ab is tested:      //
//----------------------------------------------------------------------------//
r002:      NOP 0;//Wrong action number
      S #sqSequencer.Error_Fault;
      JU k002;//Exit
_002:      NOP 0;// Action error handling
      JU k002;// Exit






NETWORK
TITLE = S002:: STEP-002:: : ACTION CODE
//================================ ACT HEADER ============================//
// ACTION ACTION ACTION ACTION ACTION ACTION ACTION ACTION ACTION ACTION  //
// AUTOCODE   AUTOCODE   AUTOCODE   AUTOCODE   AUTOCODE   AUTOCODE   AUTO //
// ACTION ACTION ACTION ACTION ACTION ACTION ACTION ACTION ACTION ACTION  //
//------------------------------------------------------------------------//
// //Action Description
aa02:      NOP 0;

  //------------------------------------------------------------------------//
  // ACT ACT ACT ACT ACT ACT ACT ACT ACT ACT ACT ACT ACT ACT ACT ACT ACT    //
  //------------------------------------------------------------------------//
      L "dbCONST".BLK.CMD.STOP;
      T #_emc_water_cmd;
      T #_emt_hex_cmd;

  //------------------------------------------------------------------------//
  // VERIFY  VERIFY VERIFY VERIFY VERIFY VERIFY VERIFY VERIFY VERIFY VERIFY //
  //------------------------------------------------------------------------//
      A(;
      L #_emc_water_state;
      L "dbCONST".BLK.STATE.STOPPED;
      ==I;
      );
      A(;
      L #_emt_hex_state;
      L "dbCONST".BLK.STATE.STOPPED;
      ==I;
      );
      S #sqSequencer.STEP.ActionVerified;//Action verified

  //------------------------------------------------------------------------//
  // Action done:                                                           //
  //------------------------------------------------------------------------//
      O #sqSequencer.STEP.ActionVerified;
      O #smc.NO_VERIFIC     ;//No verification , bypass verification code
      S #sqSequencer.STEP.ActionFinished;






  //============================= ACT FOOTER ===============================//
  // AUTOCODE   AUTOCODE   AUTOCODE   AUTOCODE   AUTOCODE   AUTOCODE   AUTO //
  // Get Ready after action finished:                                       //
  //------------------------------------------------------------------------//
      A #sqSequencer.STEP.ActionFinished;
      JCN k002;

  //------------------------------------------------------------------------//
  // Reset Action finished flag, ready for next step action:                //
  //------------------------------------------------------------------------//
      R #sqSequencer.STEP.ActionVerified;
      R #sqSequencer.STEP.ActionFinished;

  //------------------------------------------------------------------------//
  // Load Next Step Action number:                                          //
  //------------------------------------------------------------------------//
      L 02;//Load next Action
      T #sqSequencer.STEP.ActionNumber;






NETWORK
TITLE = S002:: STEP-002:: : ACTION CODE
//================================ ACT HEADER ============================//
// ACTION ACTION ACTION ACTION ACTION ACTION ACTION ACTION ACTION ACTION  //
// AUTOCODE   AUTOCODE   AUTOCODE   AUTOCODE   AUTOCODE   AUTOCODE   AUTO //
// ACTION ACTION ACTION ACTION ACTION ACTION ACTION ACTION ACTION ACTION  //
//------------------------------------------------------------------------//
// //Set emc_water to substate SETUP (Medium PW).
// //
ab02:      NOP 0;

  //------------------------------------------------------------------------//
  // ACT ACT ACT ACT ACT ACT ACT ACT ACT ACT ACT ACT ACT ACT ACT ACT ACT    //
  //------------------------------------------------------------------------//
  //Clear used flag
      SET;
      R #_prompt_connect_ok_confirm_yes;

//Set to Medium PW and start EMC2_SETUP.
      L "dbCONST".SEL.LIQUID.PW;
      T #_emc_water_medium_liquid;
      L "dbCONST".BLK.EMC2.SUBS.SETUP;
      T #_emc_water_subs;
      L "dbCONST".BLK.CMD.START;
      T #_emc_water_cmd;

  //------------------------------------------------------------------------//
  // VERIFY  VERIFY VERIFY VERIFY VERIFY VERIFY VERIFY VERIFY VERIFY VERIFY //
  //------------------------------------------------------------------------//
  //Verify if current substate changed to SETUP.
      A(;
      L #_emc_water_subs;
      L "dbCONST".BLK.EMC2.SUBS.SETUP;
      ==I;
      );
      S #sqSequencer.STEP.ActionVerified;//Action verified

  //------------------------------------------------------------------------//
  // Action done:                                                           //
  //------------------------------------------------------------------------//
      O #sqSequencer.STEP.ActionVerified;
      O #smc.NO_VERIFIC     ;//No verification , bypass verification code
      S #sqSequencer.STEP.ActionFinished;






  //============================= ACT FOOTER ===============================//
  // AUTOCODE   AUTOCODE   AUTOCODE   AUTOCODE   AUTOCODE   AUTOCODE   AUTO //
  // Get Ready after action finished:                                       //
  //------------------------------------------------------------------------//
      A #sqSequencer.STEP.ActionFinished;
      JCN k002;

  //------------------------------------------------------------------------//
  // Reset Action finished flag, ready for next step action:                //
  //------------------------------------------------------------------------//
      R #sqSequencer.STEP.ActionVerified;
      R #sqSequencer.STEP.ActionFinished;

  //------------------------------------------------------------------------//
  // Load Next Step Action number:                                          //
  //------------------------------------------------------------------------//
      L 03;//Load next Action
      T #sqSequencer.STEP.ActionNumber;






NETWORK
TITLE = S002:: STEP-002:: : ACTION CODE
//================================ ACT HEADER ============================//
// ACTION ACTION ACTION ACTION ACTION ACTION ACTION ACTION ACTION ACTION  //
// AUTOCODE   AUTOCODE   AUTOCODE   AUTOCODE   AUTOCODE   AUTOCODE   AUTO //
// ACTION ACTION ACTION ACTION ACTION ACTION ACTION ACTION ACTION ACTION  //
//------------------------------------------------------------------------//
// //Drain the heat exchanger of process cooling water
ac02:      NOP 0;

  //------------------------------------------------------------------------//
  // ACT ACT ACT ACT ACT ACT ACT ACT ACT ACT ACT ACT ACT ACT ACT ACT ACT    //
  //------------------------------------------------------------------------//
  //Set to Medium PW and start EMC2_SETUP.
      L #_r_time_hex_drain;
      T #_emt_hex_drain_time;
      L "dbCONST".BLK.EMT1.SUBS.DRAIN;
      T #_emt_hex_subs;
      L "dbCONST".BLK.CMD.START;
      T #_emt_hex_cmd;

  //------------------------------------------------------------------------//
  // VERIFY  VERIFY VERIFY VERIFY VERIFY VERIFY VERIFY VERIFY VERIFY VERIFY //
  //------------------------------------------------------------------------//
  //Verify if hex substate changed to DRAIN
      A(;
      L #_emt_hex_subs;
      L "dbCONST".BLK.EMT1.SUBS.DRAIN;
      ==I;
      );
      S #sqSequencer.STEP.ActionVerified;//Action verified

  //------------------------------------------------------------------------//
  // Action done:                                                           //
  //------------------------------------------------------------------------//
      O #sqSequencer.STEP.ActionVerified;
      O #smc.NO_VERIFIC     ;//No verification , bypass verification code
      S #sqSequencer.STEP.ActionFinished;






  //============================= STEP FOOTER ==============================//
  // AUTOCODE   AUTOCODE   AUTOCODE   AUTOCODE   AUTOCODE   AUTOCODE   AUTO //
  // Get Ready after action finished:                                       //
  //------------------------------------------------------------------------//
      A #sqSequencer.STEP.ActionFinished;
      JCN k002;

  //------------------------------------------------------------------------//
  // Reset Action finished flag, ready for next step action:                //
  //------------------------------------------------------------------------//
      R #sqSequencer.STEP.ActionVerified;
      R #sqSequencer.STEP.ActionFinished;

  //------------------------------------------------------------------------//
  // If ALL actions are finished:                                           //
  //------------------------------------------------------------------------//
      SET;
      S #sqSequencer.STEP.Finished;
      R #sqSequencer.STEP.Active;
      S #sqSequencer.STEP.Done[02];

  //------------------------------------------------------------------------//
  // End Step action(s):                                                    //
  //------------------------------------------------------------------------//
      JU k002;

//----------------------------------------------------------------------------//
// Finished Step Action(s):                                                   //
//----------------------------------------------------------------------------//
k002:      NOP 0;

      A #sqStepTimerExpired;
      S #sqSequencer.STEP.WithError[02];// Step error flag
      S #sqSequencer.Error_Fault;
      R #sqStepTimer.IN;

NETWORK
TITLE = S002:STEP-002::Begin Transition
//------------------------------------------------------------------------//
// Begin the transition code:                                             //
//------------------------------------------------------------------------//
A002:      NOP 0;
      R #sqStepTimer.IN;






  //============================= TRAN HEADER ==============================//
  // AUTOCODE   AUTOCODE   AUTOCODE   AUTOCODE   AUTOCODE   AUTOCODE   AUTO //
  // Bypass transition if manual jump:                                      //
  //------------------------------------------------------------------------//
      A #sqSequencer.STEP.Finished;
      A #smc.TRN_AND_JUMP   ;//Manual jump is set Transition as bypassed
      JCN COMM            ;//exit

NETWORK
TITLE = S002::STEP 002:TRAN 002: emc_water substate SETUP complete.
//----------------------------------------------------------------------------//
// TRAN   TRAN   TRAN   TRAN   TRAN   TRAN   TRAN   TRAN   TRAN   TRAN   TRAN //
// TRAN   TRAN   TRAN   TRAN   TRAN   TRAN   TRAN   TRAN   TRAN   TRAN   TRAN //
//----------------------------------------------------------------------------//
// emc_water substate SETUP is complete and hex draining complete.
//----------------------------------------------------------------------------//
// CONDITION   CONDITION   CONDITION   CONDITION   CONDITION   CONDITION   CO //
// CONDITION   CONDITION   CONDITION   CONDITION   CONDITION   CONDITION   CO //
//----------------------------------------------------------------------------//
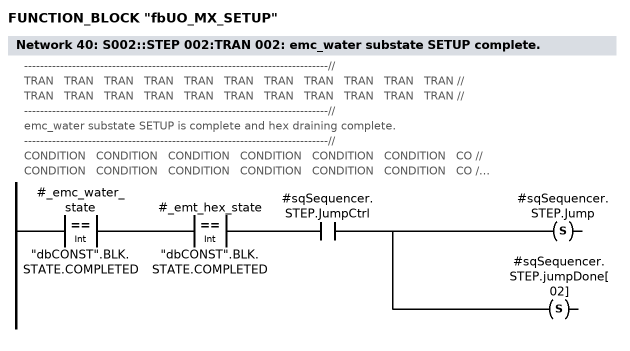
      A(;
      L #_emc_water_state;
      L "dbCONST".BLK.STATE.COMPLETED;
      ==I;
      );
      A(;
      L #_emt_hex_state;
      L "dbCONST".BLK.STATE.COMPLETED;
      ==I;
      );






  //============================= TRAN FOOTER ==============================//
  // Transition jump control:                                               //
  //------------------------------------------------------------------------//
      A #sqSequencer.STEP.JumpCtrl;
      S #sqSequencer.STEP.Jump;
      S #sqSequencer.STEP.jumpDone[02];

NETWORK
TITLE = S002:t002::TRANS-v: EXIT TRANSITION AND READY THE NEXT STEP
//------------------------------------------------------------------------//
// Check the jump flag and jump to the next step if the transition        //
// condition is true and has set the jump flag:                           //
//------------------------------------------------------------------------//
      A #sqSequencer.STEP.Jump;
      JCN x002;

      R #sqSequencer.STEP.Jump;
      R #sqSequencer.STEP.Finished;

      L 03   ;// Load next STEPNO to jump to if transition satisfied
      T #sqSequencer.STEP.NumberNext;//Next Step03.

      JU COMM            ;// Transition satisfied, Exit, go to next step
x002:      NOP 0;






NETWORK
TITLE = S002::STEP-002:EXIT TRANSITION:
//========================== STEP TRANSFER ===============================//
// Jump to the common step progression code:                              //
//------------------------------------------------------------------------//
      JU COMM;






NETWORK
TITLE = S003: STEP-03::UO_MX_SETUP : Open valves on Mx to drain flow path.
//================================ STEP HEADER ===========================//
// STEP003 STEP003 STEP003 STEP003
// AUTOCODE   AUTOCODE   AUTOCODE   AUTOCODE   AUTOCODE   AUTOCODE   AUTO //
// STEP003 STEP003 STEP003 STEP003
//------------------------------------------------------------------------//
// Open Mx outlet and MMFL transfer line valves.
//------------------------------------------------------------------------//
S003:      NOP 0;

      SET;
      R #sqSequencer.STEP.jumpDone[03];
      A #sqSequencer.CMD.Pause;//If paused jump
      JC COMM;

NETWORK
TITLE = S003:STEP-03:Begin Action

      A #sqSequencer.STEP.Finished;
      JC A003;// Exit Action code, Jump to A003 Transition code

    //----------------------------------------------------------------------//
    // Begin step Action:                                                   //
    //----------------------------------------------------------------------//
      A #sqSequencer.STEP.Active;
      JC L003;// Action number loaded, Jump to L003--Step Action List

    //----------------------------------------------------------------------//
    // Load Default/Initial Step action number:                             //
    //----------------------------------------------------------------------//
      S #sqSequencer.STEP.Active;
      S #sqStepTimer.IN;
      L 1;//First Action, Step must contain Minimum one action
      T #sqSequencer.STEP.ActionNumber;

//----------------------------------------------------------------------------//
// Step action list.                                                          //
// aann=mini Action step number(aa) inside main step number(nn)               //
// First Action aa00, Second action ab00, Third ac00, etc.                    //
//----------------------------------------------------------------------------//
L003:      NOP 0;

      L #sqSequencer.STEP.ActionNumber;
      JL r003;//Wrong Action number
      JU _003;//Action error handling
      JU aa03;//ACTION-01
      JU ab03;//ACTION-02


//----------------------------------------------------------------------------//
// More step action in the list can be inserted here, upto ab is tested:      //
//----------------------------------------------------------------------------//
r003:      NOP 0;//Wrong action number
      S #sqSequencer.Error_Fault;
      JU k003;//Exit
_003:      NOP 0;// Action error handling
      JU k003;// Exit






NETWORK
TITLE = S003:: STEP-003:: : ACTION CODE
//================================ ACT HEADER ============================//
// ACTION ACTION ACTION ACTION ACTION ACTION ACTION ACTION ACTION ACTION  //
// AUTOCODE   AUTOCODE   AUTOCODE   AUTOCODE   AUTOCODE   AUTOCODE   AUTO //
// ACTION ACTION ACTION ACTION ACTION ACTION ACTION ACTION ACTION ACTION  //
//------------------------------------------------------------------------//
// //Reset EMs
aa03:      NOP 0;

  //------------------------------------------------------------------------//
  // ACT ACT ACT ACT ACT ACT ACT ACT ACT ACT ACT ACT ACT ACT ACT ACT ACT    //
  //------------------------------------------------------------------------//
      L "dbCONST".BLK.CMD.STOP;
      T #_emv_inlet_cmd;
      T #_emv_vessel_cmd;
      T #_emx_mmfl_cmd;
      T #_emx_drain_cmd;

  //------------------------------------------------------------------------//
  // VERIFY  VERIFY VERIFY VERIFY VERIFY VERIFY VERIFY VERIFY VERIFY VERIFY //
  //------------------------------------------------------------------------//
      A(;
      L #_emv_inlet_state;
      L "dbCONST".BLK.STATE.STOPPED;
      ==I;
      );
      A(;
      L #_emv_vessel_state;
      L "dbCONST".BLK.STATE.STOPPED;
      ==I;
      );
      A(;
      L #_emx_mmfl_state;
      L "dbCONST".BLK.STATE.STOPPED;
      ==I;
      );
      A(;
      L #_emx_drain_state;
      L "dbCONST".BLK.STATE.STOPPED;
      ==I;
      );
      S #sqSequencer.STEP.ActionVerified;//Action verified

  //------------------------------------------------------------------------//
  // Action done:                                                           //
  //------------------------------------------------------------------------//
      O #sqSequencer.STEP.ActionVerified;
      O #smc.NO_VERIFIC     ;//No verification , bypass verification code
      S #sqSequencer.STEP.ActionFinished;






  //============================= ACT FOOTER ===============================//
  // AUTOCODE   AUTOCODE   AUTOCODE   AUTOCODE   AUTOCODE   AUTOCODE   AUTO //
  // Get Ready after action finished:                                       //
  //------------------------------------------------------------------------//
      A #sqSequencer.STEP.ActionFinished;
      JCN k003;

  //------------------------------------------------------------------------//
  // Reset Action finished flag, ready for next step action:                //
  //------------------------------------------------------------------------//
      R #sqSequencer.STEP.ActionVerified;
      R #sqSequencer.STEP.ActionFinished;

  //------------------------------------------------------------------------//
  // Load Next Step Action number:                                          //
  //------------------------------------------------------------------------//
      L 02;//Load next Action
      T #sqSequencer.STEP.ActionNumber;






NETWORK
TITLE = S003:: STEP-003:: : ACTION CODE
//================================ ACT HEADER ============================//
// ACTION ACTION ACTION ACTION ACTION ACTION ACTION ACTION ACTION ACTION  //
// AUTOCODE   AUTOCODE   AUTOCODE   AUTOCODE   AUTOCODE   AUTOCODE   AUTO //
// ACTION ACTION ACTION ACTION ACTION ACTION ACTION ACTION ACTION ACTION  //
//------------------------------------------------------------------------//
// //Open valves on Mx to drain flow path to drain the vessel.
// //Clear used flags.
ab03:      NOP 0;

  //------------------------------------------------------------------------//
  // ACT ACT ACT ACT ACT ACT ACT ACT ACT ACT ACT ACT ACT ACT ACT ACT ACT    //
  //------------------------------------------------------------------------//
  //Open Mx inlet valve.
      L "dbCONST".BLK.EMV2.SUBS.CHARGE;
      T #_emv_inlet_subs;
      L "dbCONST".BLK.CMD.START;
      T #_emv_inlet_cmd;

//Open Mx outlet valve.
      L "dbCONST".BLK.EMV1.SUBS.DISCHARGE;
      T #_emv_vessel_subs;
      L "dbCONST".BLK.CMD.START;
      T #_emv_vessel_cmd;

//Open MMFL valves.
      L "dbCONST".BLK.EMX1.SUBS.CIP_MX;
      T #_emx_mmfl_subs;
      L "dbCONST".BLK.CMD.START;
      T #_emx_mmfl_cmd;

//Open CIP drain valve.
      L "dbCONST".BLK.EMX4.SUBS.CIP;
      T #_emx_drain_subs;
      L "dbCONST".BLK.CMD.START;
      T #_emx_drain_cmd;

  //------------------------------------------------------------------------//
  // VERIFY  VERIFY VERIFY VERIFY VERIFY VERIFY VERIFY VERIFY VERIFY VERIFY //
  //------------------------------------------------------------------------//
      A(;
      L #_emv_inlet_subs;
      L "dbCONST".BLK.EMV2.SUBS.CHARGE;
      ==I;
      );
      A(;
      L #_emv_vessel_subs;
      L "dbCONST".BLK.EMV1.SUBS.DISCHARGE;
      ==I;
      );
      A(;
      L #_emx_mmfl_subs;
      L "dbCONST".BLK.EMX1.SUBS.CIP_MX;
      ==I;
      );
      A(;
      L #_emx_drain_subs;
      L "dbCONST".BLK.EMX4.SUBS.CIP;
      ==I;
      );
      S #sqSequencer.STEP.ActionVerified;//Action verified

  //------------------------------------------------------------------------//
  // Action done:                                                           //
  //------------------------------------------------------------------------//
      O #sqSequencer.STEP.ActionVerified;
      O #smc.NO_VERIFIC     ;//No verification , bypass verification code
      S #sqSequencer.STEP.ActionFinished;






  //============================= STEP FOOTER ==============================//
  // AUTOCODE   AUTOCODE   AUTOCODE   AUTOCODE   AUTOCODE   AUTOCODE   AUTO //
  // Get Ready after action finished:                                       //
  //------------------------------------------------------------------------//
      A #sqSequencer.STEP.ActionFinished;
      JCN k003;

  //------------------------------------------------------------------------//
  // Reset Action finished flag, ready for next step action:                //
  //------------------------------------------------------------------------//
      R #sqSequencer.STEP.ActionVerified;
      R #sqSequencer.STEP.ActionFinished;

  //------------------------------------------------------------------------//
  // If ALL actions are finished:                                           //
  //------------------------------------------------------------------------//
      SET;
      S #sqSequencer.STEP.Finished;
      R #sqSequencer.STEP.Active;
      S #sqSequencer.STEP.Done[03];

  //------------------------------------------------------------------------//
  // End Step action(s):                                                    //
  //------------------------------------------------------------------------//
      JU k003;

//----------------------------------------------------------------------------//
// Finished Step Action(s):                                                   //
//----------------------------------------------------------------------------//
k003:      NOP 0;

      A #sqStepTimerExpired;
      S #sqSequencer.STEP.WithError[03];// Step error flag
      S #sqSequencer.Error_Fault;
      R #sqStepTimer.IN;

NETWORK
TITLE = S003:STEP-003::Begin Transition
//------------------------------------------------------------------------//
// Begin the transition code:                                             //
//------------------------------------------------------------------------//
A003:      NOP 0;
      R #sqStepTimer.IN;






  //============================= TRAN HEADER ==============================//
  // AUTOCODE   AUTOCODE   AUTOCODE   AUTOCODE   AUTOCODE   AUTOCODE   AUTO //
  // Bypass transition if manual jump:                                      //
  //------------------------------------------------------------------------//
      A #sqSequencer.STEP.Finished;
      A #smc.TRN_AND_JUMP   ;//Manual jump is set Transition as bypassed
      JCN COMM            ;//exit

NETWORK
TITLE = S003::STEP 003:TRAN 003: Drain valves opened
//----------------------------------------------------------------------------//
// TRAN   TRAN   TRAN   TRAN   TRAN   TRAN   TRAN   TRAN   TRAN   TRAN   TRAN //
// TRAN   TRAN   TRAN   TRAN   TRAN   TRAN   TRAN   TRAN   TRAN   TRAN   TRAN //
//----------------------------------------------------------------------------//
// Drain path valves are opened.
//----------------------------------------------------------------------------//
// CONDITION   CONDITION   CONDITION   CONDITION   CONDITION   CONDITION   CO //
// CONDITION   CONDITION   CONDITION   CONDITION   CONDITION   CONDITION   CO //
//----------------------------------------------------------------------------//
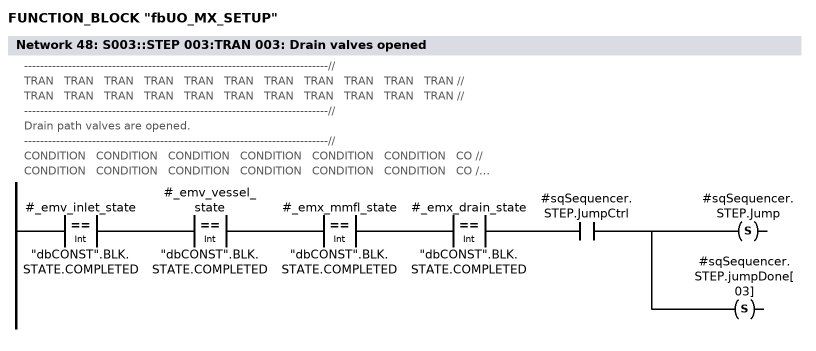
      A(;
      L #_emv_inlet_state;
      L "dbCONST".BLK.STATE.COMPLETED;
      ==I;
      );
      A(;
      L #_emv_vessel_state;
      L "dbCONST".BLK.STATE.COMPLETED;
      ==I;
      );
      A(;
      L #_emx_mmfl_state;
      L "dbCONST".BLK.STATE.COMPLETED;
      ==I;
      );
      A(;
      L #_emx_drain_state;
      L "dbCONST".BLK.STATE.COMPLETED;
      ==I;
      );






  //============================= TRAN FOOTER ==============================//
  // Transition jump control:                                               //
  //------------------------------------------------------------------------//
      A #sqSequencer.STEP.JumpCtrl;
      S #sqSequencer.STEP.Jump;
      S #sqSequencer.STEP.jumpDone[03];

NETWORK
TITLE = S003:t003::TRANS-v: EXIT TRANSITION AND READY THE NEXT STEP
//------------------------------------------------------------------------//
// Check the jump flag and jump to the next step if the transition        //
// condition is true and has set the jump flag:                           //
//------------------------------------------------------------------------//
      A #sqSequencer.STEP.Jump;
      JCN x003;

      R #sqSequencer.STEP.Jump;
      R #sqSequencer.STEP.Finished;

      L 04   ;// Load next STEPNO to jump to if transition satisfied
      T #sqSequencer.STEP.NumberNext;//Next Step04.

      JU COMM            ;// Transition satisfied, Exit, go to next step
x003:      NOP 0;






NETWORK
TITLE = S003::STEP-003:EXIT TRANSITION:
//========================== STEP TRANSFER ===============================//
// Jump to the common step progression code:                              //
//------------------------------------------------------------------------//
      JU COMM;






NETWORK
TITLE = S004: STEP-04::UO_MX_SETUP : Wait for vessel to be empty
//================================ STEP HEADER ===========================//
// STEP004 STEP004 STEP004 STEP004
// AUTOCODE   AUTOCODE   AUTOCODE   AUTOCODE   AUTOCODE   AUTOCODE   AUTO //
// STEP004 STEP004 STEP004 STEP004
//------------------------------------------------------------------------//
// Wait for vessel to drain fully
//------------------------------------------------------------------------//
S004:      NOP 0;

      SET;
      R #sqSequencer.STEP.jumpDone[04];
      A #sqSequencer.CMD.Pause;//If paused jump
      JC COMM;

NETWORK
TITLE = S004:STEP-04:Begin Action

      A #sqSequencer.STEP.Finished;
      JC A004;// Exit Action code, Jump to A004 Transition code

    //----------------------------------------------------------------------//
    // Begin step Action:                                                   //
    //----------------------------------------------------------------------//
      A #sqSequencer.STEP.Active;
      JC L004;// Action number loaded, Jump to L004--Step Action List

    //----------------------------------------------------------------------//
    // Load Default/Initial Step action number:                             //
    //----------------------------------------------------------------------//
      S #sqSequencer.STEP.Active;
      S #sqStepTimer.IN;
      L 1;//First Action, Step must contain Minimum one action
      T #sqSequencer.STEP.ActionNumber;

//----------------------------------------------------------------------------//
// Step action list.                                                          //
// aann=mini Action step number(aa) inside main step number(nn)               //
// First Action aa00, Second action ab00, Third ac00, etc.                    //
//----------------------------------------------------------------------------//
L004:      NOP 0;

      L #sqSequencer.STEP.ActionNumber;
      JL r004;//Wrong Action number
      JU _004;//Action error handling
      JU aa04;//ACTION-01


//----------------------------------------------------------------------------//
// More step action in the list can be inserted here, upto ab is tested:      //
//----------------------------------------------------------------------------//
r004:      NOP 0;//Wrong action number
      S #sqSequencer.Error_Fault;
      JU k004;//Exit
_004:      NOP 0;// Action error handling
      JU k004;// Exit






NETWORK
TITLE = S004:: STEP-004:: : ACTION CODE
//================================ ACT HEADER ============================//
// ACTION ACTION ACTION ACTION ACTION ACTION ACTION ACTION ACTION ACTION  //
// AUTOCODE   AUTOCODE   AUTOCODE   AUTOCODE   AUTOCODE   AUTOCODE   AUTO //
// ACTION ACTION ACTION ACTION ACTION ACTION ACTION ACTION ACTION ACTION  //
//------------------------------------------------------------------------//
// //
aa04:      NOP 0;

  //------------------------------------------------------------------------//
  // ACT ACT ACT ACT ACT ACT ACT ACT ACT ACT ACT ACT ACT ACT ACT ACT ACT    //
  //------------------------------------------------------------------------//


  //------------------------------------------------------------------------//
  // VERIFY  VERIFY VERIFY VERIFY VERIFY VERIFY VERIFY VERIFY VERIFY VERIFY //
  //------------------------------------------------------------------------//

      S #sqSequencer.STEP.ActionVerified;//Action verified

  //------------------------------------------------------------------------//
  // Action done:                                                           //
  //------------------------------------------------------------------------//
      O #sqSequencer.STEP.ActionVerified;
      O #smc.NO_VERIFIC     ;//No verification , bypass verification code
      S #sqSequencer.STEP.ActionFinished;






  //============================= STEP FOOTER ==============================//
  // AUTOCODE   AUTOCODE   AUTOCODE   AUTOCODE   AUTOCODE   AUTOCODE   AUTO //
  // Get Ready after action finished:                                       //
  //------------------------------------------------------------------------//
      A #sqSequencer.STEP.ActionFinished;
      JCN k004;

  //------------------------------------------------------------------------//
  // Reset Action finished flag, ready for next step action:                //
  //------------------------------------------------------------------------//
      R #sqSequencer.STEP.ActionVerified;
      R #sqSequencer.STEP.ActionFinished;

  //------------------------------------------------------------------------//
  // If ALL actions are finished:                                           //
  //------------------------------------------------------------------------//
      SET;
      S #sqSequencer.STEP.Finished;
      R #sqSequencer.STEP.Active;
      S #sqSequencer.STEP.Done[04];

  //------------------------------------------------------------------------//
  // End Step action(s):                                                    //
  //------------------------------------------------------------------------//
      JU k004;

//----------------------------------------------------------------------------//
// Finished Step Action(s):                                                   //
//----------------------------------------------------------------------------//
k004:      NOP 0;

      A #sqStepTimerExpired;
      S #sqSequencer.STEP.WithError[04];// Step error flag
      S #sqSequencer.Error_Fault;
      R #sqStepTimer.IN;

NETWORK
TITLE = S004:STEP-004::Begin Transition
//------------------------------------------------------------------------//
// Begin the transition code:                                             //
//------------------------------------------------------------------------//
A004:      NOP 0;
      R #sqStepTimer.IN;






  //============================= TRAN HEADER ==============================//
  // AUTOCODE   AUTOCODE   AUTOCODE   AUTOCODE   AUTOCODE   AUTOCODE   AUTO //
  // Bypass transition if manual jump:                                      //
  //------------------------------------------------------------------------//
      A #sqSequencer.STEP.Finished;
      A #smc.TRN_AND_JUMP   ;//Manual jump is set Transition as bypassed
      JCN COMM            ;//exit

NETWORK
TITLE = S004::STEP 004:TRAN 004: Wait for vessel empty
//----------------------------------------------------------------------------//
// TRAN   TRAN   TRAN   TRAN   TRAN   TRAN   TRAN   TRAN   TRAN   TRAN   TRAN //
// TRAN   TRAN   TRAN   TRAN   TRAN   TRAN   TRAN   TRAN   TRAN   TRAN   TRAN //
//----------------------------------------------------------------------------//
// Jump when vessel mass indicates empty
//----------------------------------------------------------------------------//
// CONDITION   CONDITION   CONDITION   CONDITION   CONDITION   CONDITION   CO //
// CONDITION   CONDITION   CONDITION   CONDITION   CONDITION   CONDITION   CO //
//----------------------------------------------------------------------------//
      A(;
      L #_emm_vessel_mi_vessel_pv;
      L 0.0;
      <=R;
      );






  //============================= TRAN FOOTER ==============================//
  // Transition jump control:                                               //
  //------------------------------------------------------------------------//
      A #sqSequencer.STEP.JumpCtrl;
      S #sqSequencer.STEP.Jump;
      S #sqSequencer.STEP.jumpDone[04];

NETWORK
TITLE = S004:t004::TRANS-v: EXIT TRANSITION AND READY THE NEXT STEP
//------------------------------------------------------------------------//
// Check the jump flag and jump to the next step if the transition        //
// condition is true and has set the jump flag:                           //
//------------------------------------------------------------------------//
      A #sqSequencer.STEP.Jump;
      JCN x004;

      R #sqSequencer.STEP.Jump;
      R #sqSequencer.STEP.Finished;

      L 05   ;// Load next STEPNO to jump to if transition satisfied
      T #sqSequencer.STEP.NumberNext;//Next Step05.

      JU COMM            ;// Transition satisfied, Exit, go to next step
x004:      NOP 0;






NETWORK
TITLE = S004::STEP-004:EXIT TRANSITION:
//========================== STEP TRANSFER ===============================//
// Jump to the common step progression code:                              //
//------------------------------------------------------------------------//
      JU COMM;






NETWORK
TITLE = S005: STEP-05::UO_MX_SETUP : Close drain valve
//================================ STEP HEADER ===========================//
// STEP005 STEP005 STEP005 STEP005
// AUTOCODE   AUTOCODE   AUTOCODE   AUTOCODE   AUTOCODE   AUTOCODE   AUTO //
// STEP005 STEP005 STEP005 STEP005
//------------------------------------------------------------------------//
// Close outlet line drain valve.
//------------------------------------------------------------------------//
S005:      NOP 0;

      SET;
      R #sqSequencer.STEP.jumpDone[05];
      A #sqSequencer.CMD.Pause;//If paused jump
      JC COMM;

NETWORK
TITLE = S005:STEP-05:Begin Action

      A #sqSequencer.STEP.Finished;
      JC A005;// Exit Action code, Jump to A005 Transition code

    //----------------------------------------------------------------------//
    // Begin step Action:                                                   //
    //----------------------------------------------------------------------//
      A #sqSequencer.STEP.Active;
      JC L005;// Action number loaded, Jump to L005--Step Action List

    //----------------------------------------------------------------------//
    // Load Default/Initial Step action number:                             //
    //----------------------------------------------------------------------//
      S #sqSequencer.STEP.Active;
      S #sqStepTimer.IN;
      L 1;//First Action, Step must contain Minimum one action
      T #sqSequencer.STEP.ActionNumber;

//----------------------------------------------------------------------------//
// Step action list.                                                          //
// aann=mini Action step number(aa) inside main step number(nn)               //
// First Action aa00, Second action ab00, Third ac00, etc.                    //
//----------------------------------------------------------------------------//
L005:      NOP 0;

      L #sqSequencer.STEP.ActionNumber;
      JL r005;//Wrong Action number
      JU _005;//Action error handling
      JU aa05;//ACTION-01


//----------------------------------------------------------------------------//
// More step action in the list can be inserted here, upto ab is tested:      //
//----------------------------------------------------------------------------//
r005:      NOP 0;//Wrong action number
      S #sqSequencer.Error_Fault;
      JU k005;//Exit
_005:      NOP 0;// Action error handling
      JU k005;// Exit






NETWORK
TITLE = S005:: STEP-005:: : ACTION CODE
//================================ ACT HEADER ============================//
// ACTION ACTION ACTION ACTION ACTION ACTION ACTION ACTION ACTION ACTION  //
// AUTOCODE   AUTOCODE   AUTOCODE   AUTOCODE   AUTOCODE   AUTOCODE   AUTO //
// ACTION ACTION ACTION ACTION ACTION ACTION ACTION ACTION ACTION ACTION  //
//------------------------------------------------------------------------//
// //Reset EMs
aa05:      NOP 0;

  //------------------------------------------------------------------------//
  // ACT ACT ACT ACT ACT ACT ACT ACT ACT ACT ACT ACT ACT ACT ACT ACT ACT    //
  //------------------------------------------------------------------------//
      L "dbCONST".BLK.CMD.STOP;
      T #_emx_drain_cmd;

  //------------------------------------------------------------------------//
  // VERIFY  VERIFY VERIFY VERIFY VERIFY VERIFY VERIFY VERIFY VERIFY VERIFY //
  //------------------------------------------------------------------------//
      A(;
      L #_emx_drain_state;
      L "dbCONST".BLK.STATE.STOPPED;
      ==I;
      );
      S #sqSequencer.STEP.ActionVerified;//Action verified

  //------------------------------------------------------------------------//
  // Action done:                                                           //
  //------------------------------------------------------------------------//
      O #sqSequencer.STEP.ActionVerified;
      O #smc.NO_VERIFIC     ;//No verification , bypass verification code
      S #sqSequencer.STEP.ActionFinished;






  //============================= STEP FOOTER ==============================//
  // AUTOCODE   AUTOCODE   AUTOCODE   AUTOCODE   AUTOCODE   AUTOCODE   AUTO //
  // Get Ready after action finished:                                       //
  //------------------------------------------------------------------------//
      A #sqSequencer.STEP.ActionFinished;
      JCN k005;

  //------------------------------------------------------------------------//
  // Reset Action finished flag, ready for next step action:                //
  //------------------------------------------------------------------------//
      R #sqSequencer.STEP.ActionVerified;
      R #sqSequencer.STEP.ActionFinished;

  //------------------------------------------------------------------------//
  // If ALL actions are finished:                                           //
  //------------------------------------------------------------------------//
      SET;
      S #sqSequencer.STEP.Finished;
      R #sqSequencer.STEP.Active;
      S #sqSequencer.STEP.Done[05];

  //------------------------------------------------------------------------//
  // End Step action(s):                                                    //
  //------------------------------------------------------------------------//
      JU k005;

//----------------------------------------------------------------------------//
// Finished Step Action(s):                                                   //
//----------------------------------------------------------------------------//
k005:      NOP 0;

      A #sqStepTimerExpired;
      S #sqSequencer.STEP.WithError[05];// Step error flag
      S #sqSequencer.Error_Fault;
      R #sqStepTimer.IN;

NETWORK
TITLE = S005:STEP-005::Begin Transition
//------------------------------------------------------------------------//
// Begin the transition code:                                             //
//------------------------------------------------------------------------//
A005:      NOP 0;
      R #sqStepTimer.IN;






  //============================= TRAN HEADER ==============================//
  // AUTOCODE   AUTOCODE   AUTOCODE   AUTOCODE   AUTOCODE   AUTOCODE   AUTO //
  // Bypass transition if manual jump:                                      //
  //------------------------------------------------------------------------//
      A #sqSequencer.STEP.Finished;
      A #smc.TRN_AND_JUMP   ;//Manual jump is set Transition as bypassed
      JCN COMM            ;//exit

NETWORK
TITLE = S005::STEP 005:TRAN 005: Empty transition
//----------------------------------------------------------------------------//
// TRAN   TRAN   TRAN   TRAN   TRAN   TRAN   TRAN   TRAN   TRAN   TRAN   TRAN //
// TRAN   TRAN   TRAN   TRAN   TRAN   TRAN   TRAN   TRAN   TRAN   TRAN   TRAN //
//----------------------------------------------------------------------------//
// Unconditional jump
//----------------------------------------------------------------------------//
// CONDITION   CONDITION   CONDITION   CONDITION   CONDITION   CONDITION   CO //
// CONDITION   CONDITION   CONDITION   CONDITION   CONDITION   CONDITION   CO //
//----------------------------------------------------------------------------//
      A "uncondJump";






  //============================= TRAN FOOTER ==============================//
  // Transition jump control:                                               //
  //------------------------------------------------------------------------//
      A #sqSequencer.STEP.JumpCtrl;
      S #sqSequencer.STEP.Jump;
      S #sqSequencer.STEP.jumpDone[05];

NETWORK
TITLE = S005:t005::TRANS-v: EXIT TRANSITION AND READY THE NEXT STEP
//------------------------------------------------------------------------//
// Check the jump flag and jump to the next step if the transition        //
// condition is true and has set the jump flag:                           //
//------------------------------------------------------------------------//
      A #sqSequencer.STEP.Jump;
      JCN x005;

      R #sqSequencer.STEP.Jump;
      R #sqSequencer.STEP.Finished;

      L 06   ;// Load next STEPNO to jump to if transition satisfied
      T #sqSequencer.STEP.NumberNext;//Next Step06.

      JU COMM            ;// Transition satisfied, Exit, go to next step
x005:      NOP 0;






NETWORK
TITLE = S005::STEP-005:EXIT TRANSITION:
//========================== STEP TRANSFER ===============================//
// Jump to the common step progression code:                              //
//------------------------------------------------------------------------//
      JU COMM;






NETWORK
TITLE = S006: STEP-06::UO_MX_SETUP : Start Vacuum
//================================ STEP HEADER ===========================//
// STEP006 STEP006 STEP006 STEP006
// AUTOCODE   AUTOCODE   AUTOCODE   AUTOCODE   AUTOCODE   AUTOCODE   AUTO //
// STEP006 STEP006 STEP006 STEP006
//------------------------------------------------------------------------//
// Enable vacuum.
// Start vacuum timer(TIME_EJECT).
// Log Vacuum begin time
//------------------------------------------------------------------------//
S006:      NOP 0;

      SET;
      R #sqSequencer.STEP.jumpDone[06];
      A #sqSequencer.CMD.Pause;//If paused jump
      JC COMM;

NETWORK
TITLE = S006:STEP-06:Begin Action

      A #sqSequencer.STEP.Finished;
      JC A006;// Exit Action code, Jump to A006 Transition code

    //----------------------------------------------------------------------//
    // Begin step Action:                                                   //
    //----------------------------------------------------------------------//
      A #sqSequencer.STEP.Active;
      JC L006;// Action number loaded, Jump to L006--Step Action List

    //----------------------------------------------------------------------//
    // Load Default/Initial Step action number:                             //
    //----------------------------------------------------------------------//
      S #sqSequencer.STEP.Active;
      S #sqStepTimer.IN;
      L 1;//First Action, Step must contain Minimum one action
      T #sqSequencer.STEP.ActionNumber;

//----------------------------------------------------------------------------//
// Step action list.                                                          //
// aann=mini Action step number(aa) inside main step number(nn)               //
// First Action aa00, Second action ab00, Third ac00, etc.                    //
//----------------------------------------------------------------------------//
L006:      NOP 0;

      L #sqSequencer.STEP.ActionNumber;
      JL r006;//Wrong Action number
      JU _006;//Action error handling
      JU aa06;//ACTION-01
      JU ab06;//ACTION-02
      JU ac06;//ACTION-03


//----------------------------------------------------------------------------//
// More step action in the list can be inserted here, upto ab is tested:      //
//----------------------------------------------------------------------------//
r006:      NOP 0;//Wrong action number
      S #sqSequencer.Error_Fault;
      JU k006;//Exit
_006:      NOP 0;// Action error handling
      JU k006;// Exit






NETWORK
TITLE = S006:: STEP-006:: : ACTION CODE
//================================ ACT HEADER ============================//
// ACTION ACTION ACTION ACTION ACTION ACTION ACTION ACTION ACTION ACTION  //
// AUTOCODE   AUTOCODE   AUTOCODE   AUTOCODE   AUTOCODE   AUTOCODE   AUTO //
// ACTION ACTION ACTION ACTION ACTION ACTION ACTION ACTION ACTION ACTION  //
//------------------------------------------------------------------------//
// //Reset gas EM
aa06:      NOP 0;

  //------------------------------------------------------------------------//
  // ACT ACT ACT ACT ACT ACT ACT ACT ACT ACT ACT ACT ACT ACT ACT ACT ACT    //
  //------------------------------------------------------------------------//
      L "dbCONST".BLK.CMD.STOP;
      T #_emc_gas_cmd;

  //------------------------------------------------------------------------//
  // VERIFY  VERIFY VERIFY VERIFY VERIFY VERIFY VERIFY VERIFY VERIFY VERIFY //
  //------------------------------------------------------------------------//
      A(;
      L #_emc_gas_state;
      L "dbCONST".BLK.STATE.STOPPED;
      ==I;
      );
      S #sqSequencer.STEP.ActionVerified;//Action verified

  //------------------------------------------------------------------------//
  // Action done:                                                           //
  //------------------------------------------------------------------------//
      O #sqSequencer.STEP.ActionVerified;
      O #smc.NO_VERIFIC     ;//No verification , bypass verification code
      S #sqSequencer.STEP.ActionFinished;






  //============================= ACT FOOTER ===============================//
  // AUTOCODE   AUTOCODE   AUTOCODE   AUTOCODE   AUTOCODE   AUTOCODE   AUTO //
  // Get Ready after action finished:                                       //
  //------------------------------------------------------------------------//
      A #sqSequencer.STEP.ActionFinished;
      JCN k006;

  //------------------------------------------------------------------------//
  // Reset Action finished flag, ready for next step action:                //
  //------------------------------------------------------------------------//
      R #sqSequencer.STEP.ActionVerified;
      R #sqSequencer.STEP.ActionFinished;

  //------------------------------------------------------------------------//
  // Load Next Step Action number:                                          //
  //------------------------------------------------------------------------//
      L 02;//Load next Action
      T #sqSequencer.STEP.ActionNumber;






NETWORK
TITLE = S006:: STEP-006:: : ACTION CODE
//================================ ACT HEADER ============================//
// ACTION ACTION ACTION ACTION ACTION ACTION ACTION ACTION ACTION ACTION  //
// AUTOCODE   AUTOCODE   AUTOCODE   AUTOCODE   AUTOCODE   AUTOCODE   AUTO //
// ACTION ACTION ACTION ACTION ACTION ACTION ACTION ACTION ACTION ACTION  //
//------------------------------------------------------------------------//
// //Enable vacuum.
// //Reset timer.
ab06:      NOP 0;

  //------------------------------------------------------------------------//
  // ACT ACT ACT ACT ACT ACT ACT ACT ACT ACT ACT ACT ACT ACT ACT ACT ACT    //
  //------------------------------------------------------------------------//
  //Enable vacuum.
      L "dbCONST".SEL.GAS.VACUUM;
      T #_emc_gas_medium_gas;
      L "dbCONST".BLK.EMC1.SUBS.VALVE;
      T #_emc_gas_subs;
      L "dbCONST".BLK.CMD.START;
      T #_emc_gas_cmd;

// Reset vacuum timer
      R #sqSeqTimerStart;

  //------------------------------------------------------------------------//
  // VERIFY  VERIFY VERIFY VERIFY VERIFY VERIFY VERIFY VERIFY VERIFY VERIFY //
  //------------------------------------------------------------------------//
      AN #SQ_TIMER.Q;
      S #sqSequencer.STEP.ActionVerified;//Action verified

  //------------------------------------------------------------------------//
  // Action done:                                                           //
  //------------------------------------------------------------------------//
      O #sqSequencer.STEP.ActionVerified;
      O #smc.NO_VERIFIC     ;//No verification , bypass verification code
      S #sqSequencer.STEP.ActionFinished;






  //============================= ACT FOOTER ===============================//
  // AUTOCODE   AUTOCODE   AUTOCODE   AUTOCODE   AUTOCODE   AUTOCODE   AUTO //
  // Get Ready after action finished:                                       //
  //------------------------------------------------------------------------//
      A #sqSequencer.STEP.ActionFinished;
      JCN k006;

  //------------------------------------------------------------------------//
  // Reset Action finished flag, ready for next step action:                //
  //------------------------------------------------------------------------//
      R #sqSequencer.STEP.ActionVerified;
      R #sqSequencer.STEP.ActionFinished;

  //------------------------------------------------------------------------//
  // Load Next Step Action number:                                          //
  //------------------------------------------------------------------------//
      L 03;//Load next Action
      T #sqSequencer.STEP.ActionNumber;






NETWORK
TITLE = S006:: STEP-006:: : ACTION CODE
//================================ ACT HEADER ============================//
// ACTION ACTION ACTION ACTION ACTION ACTION ACTION ACTION ACTION ACTION  //
// AUTOCODE   AUTOCODE   AUTOCODE   AUTOCODE   AUTOCODE   AUTOCODE   AUTO //
// ACTION ACTION ACTION ACTION ACTION ACTION ACTION ACTION ACTION ACTION  //
//------------------------------------------------------------------------//
// //Start vacuum timer. Log Vacuum begin time
ac06:      NOP 0;

  //------------------------------------------------------------------------//
  // ACT ACT ACT ACT ACT ACT ACT ACT ACT ACT ACT ACT ACT ACT ACT ACT ACT    //
  //------------------------------------------------------------------------//
      L #_r_time_eject;
      T #SQ_TIMER.PT;
      S #sqSeqTimerStart;

//Log vacuum begin time
      SET;
      S #_log_msg_vacuum_begin;

  //------------------------------------------------------------------------//
  // VERIFY  VERIFY VERIFY VERIFY VERIFY VERIFY VERIFY VERIFY VERIFY VERIFY //
  //------------------------------------------------------------------------//
      A #sqSeqTimerStart;
      S #sqSequencer.STEP.ActionVerified;//Action verified

  //------------------------------------------------------------------------//
  // Action done:                                                           //
  //------------------------------------------------------------------------//
      O #sqSequencer.STEP.ActionVerified;
      O #smc.NO_VERIFIC     ;//No verification , bypass verification code
      S #sqSequencer.STEP.ActionFinished;






  //============================= STEP FOOTER ==============================//
  // AUTOCODE   AUTOCODE   AUTOCODE   AUTOCODE   AUTOCODE   AUTOCODE   AUTO //
  // Get Ready after action finished:                                       //
  //------------------------------------------------------------------------//
      A #sqSequencer.STEP.ActionFinished;
      JCN k006;

  //------------------------------------------------------------------------//
  // Reset Action finished flag, ready for next step action:                //
  //------------------------------------------------------------------------//
      R #sqSequencer.STEP.ActionVerified;
      R #sqSequencer.STEP.ActionFinished;

  //------------------------------------------------------------------------//
  // If ALL actions are finished:                                           //
  //------------------------------------------------------------------------//
      SET;
      S #sqSequencer.STEP.Finished;
      R #sqSequencer.STEP.Active;
      S #sqSequencer.STEP.Done[06];

  //------------------------------------------------------------------------//
  // End Step action(s):                                                    //
  //------------------------------------------------------------------------//
      JU k006;

//----------------------------------------------------------------------------//
// Finished Step Action(s):                                                   //
//----------------------------------------------------------------------------//
k006:      NOP 0;

      A #sqStepTimerExpired;
      S #sqSequencer.STEP.WithError[06];// Step error flag
      S #sqSequencer.Error_Fault;
      R #sqStepTimer.IN;

NETWORK
TITLE = S006:STEP-006::Begin Transition
//------------------------------------------------------------------------//
// Begin the transition code:                                             //
//------------------------------------------------------------------------//
A006:      NOP 0;
      R #sqStepTimer.IN;






  //============================= TRAN HEADER ==============================//
  // AUTOCODE   AUTOCODE   AUTOCODE   AUTOCODE   AUTOCODE   AUTOCODE   AUTO //
  // Bypass transition if manual jump:                                      //
  //------------------------------------------------------------------------//
      A #sqSequencer.STEP.Finished;
      A #smc.TRN_AND_JUMP   ;//Manual jump is set Transition as bypassed
      JCN COMM            ;//exit

NETWORK
TITLE = S006::STEP 006:TRAN 006: Timer expired?
//----------------------------------------------------------------------------//
// TRAN   TRAN   TRAN   TRAN   TRAN   TRAN   TRAN   TRAN   TRAN   TRAN   TRAN //
// TRAN   TRAN   TRAN   TRAN   TRAN   TRAN   TRAN   TRAN   TRAN   TRAN   TRAN //
//----------------------------------------------------------------------------//
// Vacuum timer expired.
//----------------------------------------------------------------------------//
// CONDITION   CONDITION   CONDITION   CONDITION   CONDITION   CONDITION   CO //
// CONDITION   CONDITION   CONDITION   CONDITION   CONDITION   CONDITION   CO //
//----------------------------------------------------------------------------//
      A #SQ_TIMER.Q;






  //============================= TRAN FOOTER ==============================//
  // Transition jump control:                                               //
  //------------------------------------------------------------------------//
      A #sqSequencer.STEP.JumpCtrl;
      S #sqSequencer.STEP.Jump;
      S #sqSequencer.STEP.jumpDone[06];

NETWORK
TITLE = S006:t006::TRANS-v: EXIT TRANSITION AND READY THE NEXT STEP
//------------------------------------------------------------------------//
// Check the jump flag and jump to the next step if the transition        //
// condition is true and has set the jump flag:                           //
//------------------------------------------------------------------------//
      A #sqSequencer.STEP.Jump;
      JCN x006;

      R #sqSequencer.STEP.Jump;
      R #sqSequencer.STEP.Finished;

      L 07   ;// Load next STEPNO to jump to if transition satisfied
      T #sqSequencer.STEP.NumberNext;//Next Step07.

      JU COMM            ;// Transition satisfied, Exit, go to next step
x006:      NOP 0;






  //============================= TRAN HEADER ==============================//
  // AUTOCODE   AUTOCODE   AUTOCODE   AUTOCODE   AUTOCODE   AUTOCODE   AUTO //
  // Bypass transition if manual jump:                                      //
  //------------------------------------------------------------------------//
      A #sqSequencer.STEP.Finished;
      A #smc.TRN_AND_JUMP   ;//Manual jump is set Transition as bypassed
      JCN COMM            ;//exit

